{attribute 'qualified_only'}
{attribute 'strict'}
TYPE TGControllerMode :
(
	IControl,
	PControl
);
END_TYPE

(* stored: Version 1.1.0.1, ProductVersion 3.1.4024.12
   DUT TGControllerMode: Id {39624550-fd03-4493-b985-5d7a1c72699e} *)
